PROGRAM README
VAR
END_VAR

(*
//============
NAMING INPUTS USING UNION:
	Give Inputs/Outputs Specific Labels In: 
		DUT/INPUT_LABELS
		DUT/OUTPUT_LABELS
	
	Thus inputs have clear names and address:  
		IN._I._Label.Door_Sensor1
		
	IO is received into Array, and every input is then given a specific Label through Union. 
	IO can still be referenced in array form:
		IN._I.bArray[1];
	Because DUT/Union simply slaps a label on top of bArray[1..32], Door_Sensor1 and bArray[8] are the same thing and thus activate simultaneously.

//============
GATO E PERRO 
	Original idea of this demo project is to showcase and test different inputs, outputs and controls of PLC. Some features are needlessly complicated 
	considering the task, but are used for learning purposes. Several components are scavenged and repurposed, thus giving a but amateurish
	and hacky look to the project, but I still made an effort for professional finish.	

	Name is in Spanish to clearly distinguish test project from actual customer project. Future database names et al continue the same namoing
	convention to make it easier to copy/paste and change variables and names.
	
	End result of project is a cat figure running from dog figure, with magnetic and light sensor observing them.
	Distinguishing cat from a dog can be achieved in many ways, and I chose a middle ground between practicality, budget and reliability.
	Cat figure has a magnet glued behind it, thus "priming" the light sensor 
	-> next time a figure passes light sensor, its a cat. 
	-> If light sensor is not primed, its a dog.
	
	Inside the cabinet exists analog temperature sensor, a multiple port relay and green signal light.
 
	Cat and dog are running on electric motor, which is controlled by Vacon VFD.
	Due to availability, budget and preference, Vacon doesnt have any fancy input modules and is controlled with simple IO-pins. 
	Future learning potential is definitely there.

	 
=====================
	
	

*)

END_PROGRAM

(* stored: Version 1.1.0.1, ProductVersion 3.1.4024.10
   POU README: Id {21aadffe-44b8-4b9a-bc6a-db6fda072069}, SpecialFunc None *)
